TYPE ST_FlowControlCommands :
STRUCT
	resetCo2Consumption : BOOL;
	startMovingAvgCalculation : BOOL;
	enableFlowMpc : BOOL;
	flowSetpoint : REAL;
END_STRUCT
END_TYPE

(* stored: Version 1.1.0.1, ProductVersion 3.1.4024.9
   DUT ST_FlowControlCommands: Id {ea092267-46ff-4397-9bc8-8d38280c10af} *)
